(* IEC 61131-3 sources: tianxianzhuantaiPLC/plc/src, 5 files *)

(* ---- Turntable_Constants.st ---- *)
(******************************************************************************
  AutoShop LiteST reference source -- create this as a global constant table.
  Bind only INT wire words to D registers; keep DINT/REAL process values unbound.
******************************************************************************)
VAR_GLOBAL CONSTANT
    (* Modbus wire-register addresses; plc/register-map.md is normative. *)
    D0000_MODE : INT := 0; D0001_DIRECTION : INT := 1;
    D0002_SPEED_INDEX : INT := 2; D0003_START_SEQ : INT := 3;
    D0004_STOP_SEQ : INT := 4; D0005_SET_ZERO_SEQ : INT := 5;
    D0006_RESET_FAULT_SEQ : INT := 6; D0007_POWER_SEQ : INT := 7;
    D0008_HEARTBEAT : INT := 8; D0009_BUFFER_ACK_SEQ : INT := 9;
    D0010_TOTAL_RATIO_HI : INT := 10; D0011_TOTAL_RATIO_LO : INT := 11;
    D0012_ACCEL_HI : INT := 12; D0013_ACCEL_LO : INT := 13;
    D0014_DECEL_HI : INT := 14; D0015_DECEL_LO : INT := 15;
    D0016_STOP_DECEL_HI : INT := 16; D0017_STOP_DECEL_LO : INT := 17;
    D0018_BACKLASH_HI : INT := 18; D0019_BACKLASH_LO : INT := 19;
    D0100_RUN_STATE : INT := 100; D0101_STATUS_FLAGS : INT := 101;
    D0102_FAULT_CODE : INT := 102; D0103_POSITION_HI : INT := 103;
    D0104_POSITION_LO : INT := 104; D0105_TARGET_HI : INT := 105;
    D0106_TARGET_LO : INT := 106; D0107_VELOCITY_HI : INT := 107;
    D0108_VELOCITY_LO : INT := 108; D0109_HEARTBEAT_ECHO : INT := 109;
    D0110_START_ACK_SEQ : INT := 110; D0111_STOP_ACK_SEQ : INT := 111;
    D0112_SET_ZERO_ACK_SEQ : INT := 112; D0113_RESET_FAULT_ACK_SEQ : INT := 113;
    D0114_POWER_ACK_SEQ : INT := 114; D0115_BUFFER_ACKED_SEQ : INT := 115;
    D0116_EVENT_COUNT : INT := 116; D0117_EVENT_GENERATION : INT := 117;
    D0118_RUN_STATUS : INT := 118; D0119_RUN_START_TICK_HI : INT := 119;
    D0120_RUN_START_TICK_LO : INT := 120;
    D0200_PROTOCOL_VERSION : INT := 200; D0201_WORD_ORDER_HI : INT := 201;
    D0202_WORD_ORDER_LO : INT := 202; D0203_TIME_SYNC_REQUEST_SEQ : INT := 203;
    D0204_TICK_HI : INT := 204; D0205_TICK_LO : INT := 205;
    D0206_TIME_SYNC_RESPONSE_SEQ : INT := 206;
    D2000_EVENT_BASE : INT := 2000; D4159_EVENT_END : INT := 4159;

    MODE_MANUAL : INT := 0; MODE_AUTO : INT := 1;
    DIRECTION_CW : INT := 1; DIRECTION_CCW : INT := -1;
    STATE_INITIALIZING : INT := 0; STATE_ZERO_REQUIRED : INT := 1;
    STATE_READY : INT := 2; STATE_MANUAL_RUNNING : INT := 3;
    STATE_AUTO_RUNNING : INT := 4; STATE_STOPPING : INT := 5;
    STATE_AUTO_ABORTED : INT := 6; STATE_FAULT : INT := 7;
    RUN_IDLE : INT := 0; RUN_RUNNING : INT := 1; RUN_COMPLETED : INT := 2;
    RUN_MANUAL_STOPPED : INT := 3; RUN_AUTO_ABORTED : INT := 4;
    RUN_COMMUNICATION_ABORTED : INT := 5; RUN_FAULTED : INT := 6;
    FAULT_NONE : INT := 0; FAULT_INVALID_COMMAND : INT := 1;
    FAULT_ZERO_INTERLOCK : INT := 2; FAULT_AUTO_LIMIT : INT := 3;
    FAULT_MOTION : INT := 4; FAULT_POSITION_READ : INT := 5;
    FAULT_VELOCITY_READ : INT := 6; FAULT_HEARTBEAT : INT := 7;
    FAULT_STOP_UNSAFE : INT := 8; FAULT_AXIS_CONFIG : INT := 9;
    FAULT_START_REJECTED : INT := 10; FAULT_RESET : INT := 11;

    STATUS_ZERO_VALID : INT := 1; STATUS_POWERED : INT := 2;
    STATUS_SOFT_LIMIT : INT := 4; STATUS_BUFFER_READY : INT := 8;
    STATUS_HEARTBEAT_OK : INT := 16;
    PROTOCOL_VERSION : INT := 2;
    WORD_ORDER_PROBE_HIGH : INT := 4660; WORD_ORDER_PROBE_LOW : INT := 22136;
    TOTAL_RATIO_MILLI : DINT := 50000; (* 50.000:1 *)
    SPEED_1_DEG_S : REAL := 1.0; SPEED_2_DEG_S : REAL := 2.0;
    SPEED_3_DEG_S : REAL := 4.0; SPEED_4_DEG_S : REAL := 5.0;
    SPEED_5_DEG_S : REAL := 10.0;
    ACCELERATION_DEG_S2 : REAL := 5.0; DECELERATION_DEG_S2 : REAL := 5.0;
    SOFTWARE_STOP_DECEL_DEG_S2 : REAL := 10.0;
    ACCELERATION_MILLI_DEG_S2 : DINT := 5000;
    DECELERATION_MILLI_DEG_S2 : DINT := 5000;
    SOFTWARE_STOP_DECEL_MILLI_DEG_S2 : DINT := 10000;
    SOFT_LIMIT_MIN_DEG : REAL := -360.0; SOFT_LIMIT_MAX_DEG : REAL := 360.0;
    AUTO_DISTANCE_DEG : REAL := 360.0;
    HEARTBEAT_TIMEOUT_SCANS : INT := 1000;
    EVENT_CAPACITY : INT := 360; EVENT_RECORD_WORDS : INT := 6;
    EVENT_WORD_COUNT : INT := 2160; EVENT_MAX_CROSSINGS_PER_SCAN : INT := 360;
END_VAR

(* Create this as the sole global MODBUS_D variable table and bind addresses
   here. PRG_MAIN consumes these globals; do not redeclare them locally. *)
VAR_GLOBAL
    iD0000Mode, iD0001Direction, iD0002SpeedIndex : INT;
    iD0003StartSeq, iD0004StopSeq, iD0005SetZeroSeq, iD0006ResetFaultSeq : INT;
    iD0007PowerSeq, iD0008Heartbeat, iD0009BufferAckSeq : INT;
    iD0010RatioHi, iD0011RatioLo, iD0012AccelHi, iD0013AccelLo : INT;
    iD0014DecelHi, iD0015DecelLo, iD0016StopDecelHi, iD0017StopDecelLo : INT;
    iD0018BacklashHi, iD0019BacklashLo : INT;
    iD0100RunState, iD0101StatusFlags, iD0102FaultCode : INT;
    iD0103PositionHi, iD0104PositionLo, iD0105TargetHi, iD0106TargetLo : INT;
    iD0107VelocityHi, iD0108VelocityLo, iD0109HeartbeatEcho : INT;
    iD0110StartAck, iD0111StopAck, iD0112SetZeroAck, iD0113ResetFaultAck : INT;
    iD0114PowerAck, iD0115BufferAcked, iD0116EventCount, iD0117Generation : INT;
    iD0118RunStatus, iD0119RunStartTickHi, iD0120RunStartTickLo : INT;
    iD0200ProtocolVersion, iD0201WordOrderHi, iD0202WordOrderLo : INT;
    iD0203TimeSyncRequest, iD0204TickHi, iD0205TickLo, iD0206TimeSyncResponse : INT;
    aD2000Events : ARRAY[0..2159] OF INT;
END_VAR

(* ---- Turntable_RegisterCodec.st ---- *)
(******************************************************************************
  AutoShop LiteST reference source -- create these two FCs before the FBs.
  DINT values are always explicitly represented as high-word then low-word INTs.
  Read and verify D0201:D0202 (0x1234/0x5678) on the actual PLC before any
  hardware write.  Do not rely on a native DINT variable-table binding order.
******************************************************************************)
FUNCTION FC_DecodeI32 : DINT
VAR_INPUT
    iHighWord : INT;
    iLowWord : INT;
END_VAR
VAR
    diLowWord : DINT;
END_VAR
diLowWord := INT_TO_DINT(iLowWord);
IF diLowWord < 0 THEN diLowWord := diLowWord + 65536; END_IF;
FC_DecodeI32 := INT_TO_DINT(iHighWord) * 65536 + diLowWord;
END_FUNCTION

FUNCTION FC_SplitI32 : BOOL
VAR_INPUT
    diValue : DINT;
END_VAR
VAR_OUTPUT
    iHighWord : INT;
    iLowWord : INT;
END_VAR
VAR
    diHighWord : DINT;
    diLowWord : DINT;
END_VAR
diHighWord := diValue / 65536;
diLowWord := diValue MOD 65536;
IF diLowWord < 0 THEN
    diLowWord := diLowWord + 65536;
    diHighWord := diHighWord - 1;
END_IF;
IF diHighWord >= 32768 THEN diHighWord := diHighWord - 65536; END_IF;
IF diLowWord >= 32768 THEN diLowWord := diLowWord - 65536; END_IF;
iHighWord := DINT_TO_INT(diHighWord);
iLowWord := DINT_TO_INT(diLowWord);
FC_SplitI32 := TRUE;
END_FUNCTION

FUNCTION FC_SplitU32 : BOOL
VAR_INPUT
    diValue : DINT;
END_VAR
VAR_OUTPUT
    iHighWord : INT;
    iLowWord : INT;
END_VAR
VAR
    diHighWord : DINT;
    diLowWord : DINT;
END_VAR
diHighWord := diValue / 65536;
diLowWord := diValue MOD 65536;
IF diLowWord < 0 THEN
    diLowWord := diLowWord + 65536;
    diHighWord := diHighWord - 1;
END_IF;
IF diHighWord >= 32768 THEN diHighWord := diHighWord - 65536; END_IF;
IF diLowWord >= 32768 THEN diLowWord := diLowWord - 65536; END_IF;
iHighWord := DINT_TO_INT(diHighWord);
iLowWord := DINT_TO_INT(diLowWord);
FC_SplitU32 := TRUE;
END_FUNCTION

(* ---- FB_DegreeLogger.st ---- *)
(******************************************************************************
  AutoShop LiteST reference source -- create FB_DegreeLogger, paste declaration
  and body.  aEventWords is the INT[2160] variable-table array bound at D2000.
******************************************************************************)
FUNCTION_BLOCK FB_DegreeLogger
VAR_INPUT
    rPreviousPositionDeg : REAL;
    rCurrentPositionDeg : REAL;
    rRunOriginDeg : REAL;
    iDirection : INT;
    udiRunStartTickMs : UDINT;
    udiNowTickMs : UDINT;
    bRunStarted : BOOL;
    bRunFinished : BOOL;
    bBufferAckEdge : BOOL;
END_VAR
VAR_IN_OUT
    aEventWords : ARRAY[0..2159] OF INT;
END_VAR
VAR_OUTPUT
    bBufferReady : BOOL;
    uiEventCount : UINT;
    uiGeneration : UINT;
END_VAR
VAR
    rPreviousTravel : REAL;
    rCurrentTravel : REAL;
    rCrossingPosition : REAL;
    iFirstAngle : INT;
    iLastAngle : INT;
    iCrossing : INT;
    iTravelAngle : INT;
    iBase : INT;
    diPositionMdeg : DINT;
    udiElapsedMs : UDINT;
    iPositionHigh : INT;
    iPositionLow : INT;
    iElapsedHigh : INT;
    iElapsedLow : INT;
END_VAR

(* An acknowledged completed buffer is released before a possible run start. *)
IF bBufferAckEdge AND bBufferReady THEN
    bBufferReady := FALSE;
    uiEventCount := 0;
END_IF;

IF bRunStarted AND NOT bBufferReady THEN
    uiEventCount := 0;
    uiGeneration := uiGeneration + 1;
END_IF;

(* A sealed buffer is immutable. A controller prevents another run until ACK. *)
IF NOT bBufferReady AND NOT bRunStarted THEN
    rPreviousTravel := (rPreviousPositionDeg - rRunOriginDeg) * REAL(iDirection);
    rCurrentTravel := (rCurrentPositionDeg - rRunOriginDeg) * REAL(iDirection);
    iFirstAngle := MAX(1, REAL_TO_INT(FLOOR(rPreviousTravel)) + 1);
    iLastAngle := MIN(360, REAL_TO_INT(FLOOR(rCurrentTravel)));

    (* Fixed guard: at most 360 legal travel-angle writes per scan. *)
    FOR iCrossing := 1 TO 360 DO
        iTravelAngle := iFirstAngle + iCrossing - 1;
        IF iTravelAngle > iLastAngle THEN
            EXIT;
        END_IF;
        IF uiEventCount < 360 THEN
            iBase := 6 * uiEventCount;
            rCrossingPosition := rRunOriginDeg + REAL(iDirection) * REAL(iTravelAngle);
            diPositionMdeg := REAL_TO_DINT(rCrossingPosition * 1000.0);
            (* UDINT subtraction intentionally handles the 49.7-day tick wrap. *)
            udiElapsedMs := udiNowTickMs - udiRunStartTickMs;
            FC_SplitI32(diValue := diPositionMdeg, iHighWord => iPositionHigh, iLowWord => iPositionLow);
            FC_SplitU32(udiValue := udiElapsedMs, iHighWord => iElapsedHigh, iLowWord => iElapsedLow);
            aEventWords[iBase + 0] := INT(uiEventCount + 1);
            aEventWords[iBase + 1] := iTravelAngle;
            aEventWords[iBase + 2] := iPositionHigh;
            aEventWords[iBase + 3] := iPositionLow;
            aEventWords[iBase + 4] := iElapsedHigh;
            aEventWords[iBase + 5] := iElapsedLow;
            uiEventCount := uiEventCount + 1;
        ELSE
            EXIT;
        END_IF;
    END_FOR;
END_IF;

IF bRunFinished THEN
    bBufferReady := TRUE;
END_IF;
END_FUNCTION_BLOCK

(* ---- FB_TurntableControl.st ---- *)
(******************************************************************************
  AutoShop LiteST reference -- create FB_TurntableControl then paste it.
  It is deterministic: a commanded move remains active until MC_Stop confirms
  standstill. The heartbeat is a communication watchdog, not safety-rated.
******************************************************************************)
FUNCTION_BLOCK FB_TurntableControl
VAR_INPUT
    uiMode : UINT; iDirection : INT; uiSpeedIndex : UINT;
    uiStartSeq : UINT; uiStopSeq : UINT; uiSetZeroSeq : UINT;
    uiResetFaultSeq : UINT; uiPowerSeq : UINT; uiHeartbeat : UINT;
    uiBufferAckSeq : UINT; udiNowTickMs : UDINT;
    diTotalRatioMilli : DINT; diRequestedAccelMilli : DINT;
    diRequestedDecelMilli : DINT; diRequestedStopDecelMilli : DINT;
    diBacklashMilli : DINT;
    rActualPositionDeg : REAL; rActualVelocityDegS : REAL;
    bPositionValid : BOOL; bVelocityValid : BOOL;
    bPositionReadError : BOOL; bVelocityReadError : BOOL;
    bPowerStatus : BOOL; bPowerError : BOOL; bMoveDone : BOOL;
    bMoveBusy : BOOL; bMoveAborted : BOOL; bMoveError : BOOL;
    bStopDone : BOOL; bStopBusy : BOOL; bStopError : BOOL;
    bSetPositionDone : BOOL; bSetPositionError : BOOL;
    bResetDone : BOOL; bResetBusy : BOOL; bResetError : BOOL;
    bLoggerBufferReady : BOOL; uiLoggerEventCount : UINT;
END_VAR
VAR_OUTPUT
    bPowerEnable : BOOL; bMoveRequest : BOOL; bStopRequest : BOOL;
    bSetZeroRequest : BOOL; bResetRequest : BOOL;
    bRunStarted : BOOL; bRunFinished : BOOL; bBufferAckEdge : BOOL;
    rMoveDistance : REAL; rSelectedVelocity : REAL;
    rAcceleration : REAL; rDeceleration : REAL; rStopDeceleration : REAL;
    rRunOriginDeg : REAL; iRunDirection : INT; udiRunStartTickMs : UDINT;
    rAcceptedTargetDeg : REAL;
    uiRunState : UINT; uiRunStatus : UINT; uiFaultCode : UINT;
    uiStatusFlags : UINT; uiHeartbeatEcho : UINT;
    uiStartAckSeq : UINT; uiStopAckSeq : UINT; uiSetZeroAckSeq : UINT;
    uiResetFaultAckSeq : UINT; uiPowerAckSeq : UINT; uiBufferAckedSeq : UINT;
    uiRetainedStopReason : UINT; bUnsafeStopFailure : BOOL;
END_VAR
VAR RETAIN
    bZeroValid : BOOL;
    uiRetainedStopReasonNv : UINT;
END_VAR
VAR
    uiLastHeartbeat : UINT; uiHeartbeatAgeScans : UINT;
    bActiveRun : BOOL; bStopLatched : BOOL; bFaultStopPending : BOOL;
    uiPendingFaultCode : UINT; bPowerCommandValue : BOOL;
    bResetPending : BOOL; uiResetPendingSeq : UINT;
    bStartAccepted : BOOL;
    rCandidateTargetDeg : REAL;
END_VAR

(* Defaults are one-scan rising-edge request pulses. *)
bMoveRequest := FALSE; bStopRequest := FALSE; bSetZeroRequest := FALSE;
bResetRequest := FALSE; bRunStarted := FALSE; bRunFinished := FALSE;
bBufferAckEdge := FALSE;

IF uiRunState = STATE_INITIALIZING THEN
    IF bZeroValid THEN uiRunState := STATE_READY; ELSE uiRunState := STATE_ZERO_REQUIRED; END_IF;
END_IF;

IF uiHeartbeat <> uiLastHeartbeat THEN
    uiLastHeartbeat := uiHeartbeat; uiHeartbeatAgeScans := 0; uiHeartbeatEcho := uiHeartbeat;
ELSIF uiHeartbeatAgeScans < 65535 THEN
    uiHeartbeatAgeScans := uiHeartbeatAgeScans + 1;
END_IF;

(* Terminal Stop response is handled before accepting another command. *)
IF bStopError AND bStopLatched THEN
    (* Unsafe terminal path: motion stop was not confirmed. Inhibit power and
       keep the event buffer unsealed for on-site assessment; do not auto-retry. *)
    bActiveRun := FALSE; bStopLatched := FALSE; bUnsafeStopFailure := TRUE;
    uiRunState := STATE_FAULT; uiRunStatus := RUN_FAULTED; uiFaultCode := FAULT_STOP_UNSAFE;
    uiRetainedStopReason := RUN_FAULTED; uiRetainedStopReasonNv := RUN_FAULTED;
ELSIF bStopDone AND bActiveRun THEN
    bActiveRun := FALSE; bStopLatched := FALSE; bRunFinished := TRUE;
    IF bFaultStopPending THEN
        bFaultStopPending := FALSE; uiRunState := STATE_FAULT; uiRunStatus := RUN_FAULTED;
        uiFaultCode := uiPendingFaultCode; rAcceptedTargetDeg := rActualPositionDeg;
    ELSE
        uiRunState := STATE_READY; uiRunStatus := uiRetainedStopReason;
        rAcceptedTargetDeg := rActualPositionDeg;
    END_IF;
END_IF;

(* RESET is an axis instruction result, not a display-only flag clear. *)
IF bResetPending AND (bResetDone OR bResetError) THEN
    uiResetFaultAckSeq := uiResetPendingSeq; bResetPending := FALSE;
    IF bResetDone THEN
        uiFaultCode := FAULT_NONE; uiRunStatus := RUN_IDLE;
        bFaultStopPending := FALSE; uiPendingFaultCode := FAULT_NONE;
        bStopLatched := FALSE; bUnsafeStopFailure := FALSE;
        uiRetainedStopReason := RUN_IDLE; uiRetainedStopReasonNv := RUN_IDLE;
        IF bZeroValid THEN uiRunState := STATE_READY; ELSE uiRunState := STATE_ZERO_REQUIRED; END_IF;
    ELSE
        uiRunState := STATE_FAULT; uiRunStatus := RUN_FAULTED; uiFaultCode := FAULT_RESET;
    END_IF;
END_IF;

(* STOP_SEQ is first and also consumes a same/earlier START_SEQ. *)
IF uiStopSeq <> uiStopAckSeq THEN
    uiStopAckSeq := uiStopSeq;
    uiStartAckSeq := uiStartSeq; (* discard pending start; stop has priority *)
    IF bActiveRun AND NOT bStopLatched THEN
        bStopLatched := TRUE; bStopRequest := TRUE; uiRunState := STATE_STOPPING;
        IF uiMode = MODE_AUTO THEN uiRetainedStopReason := RUN_AUTO_ABORTED;
        ELSE uiRetainedStopReason := RUN_MANUAL_STOPPED; END_IF;
        uiRetainedStopReasonNv := uiRetainedStopReason; uiRunStatus := uiRetainedStopReason;
    END_IF;
ELSIF bActiveRun AND NOT bStopLatched AND
      (bPositionReadError OR bVelocityReadError OR NOT bPositionValid OR NOT bVelocityValid
       OR bPowerError OR bMoveError OR bMoveAborted) THEN
    (* Preserve active motion and command MC_Stop in this scan; only Done seals it. *)
    bStopLatched := TRUE; bFaultStopPending := TRUE; bStopRequest := TRUE;
    uiRunState := STATE_STOPPING; uiRunStatus := RUN_FAULTED;
    uiRetainedStopReason := RUN_FAULTED; uiRetainedStopReasonNv := RUN_FAULTED;
    IF bPositionReadError OR NOT bPositionValid THEN uiPendingFaultCode := FAULT_POSITION_READ;
    ELSIF bVelocityReadError OR NOT bVelocityValid THEN uiPendingFaultCode := FAULT_VELOCITY_READ;
    ELSE uiPendingFaultCode := FAULT_MOTION; END_IF;
ELSIF bActiveRun AND NOT bStopLatched AND (uiHeartbeatAgeScans > 1000) THEN
    bStopLatched := TRUE; bStopRequest := TRUE; uiRunState := STATE_STOPPING;
    uiRetainedStopReason := RUN_COMMUNICATION_ABORTED;
    uiRetainedStopReasonNv := uiRetainedStopReason; uiRunStatus := RUN_COMMUNICATION_ABORTED;
    uiFaultCode := FAULT_HEARTBEAT;
ELSIF uiResetFaultSeq <> uiResetFaultAckSeq AND NOT bResetPending THEN
    IF bActiveRun THEN
        uiResetFaultAckSeq := uiResetFaultSeq; uiFaultCode := FAULT_INVALID_COMMAND;
    ELSE
        bResetPending := TRUE; uiResetPendingSeq := uiResetFaultSeq; bResetRequest := TRUE;
    END_IF;
ELSIF uiBufferAckSeq <> uiBufferAckedSeq THEN
    IF NOT bActiveRun THEN uiBufferAckedSeq := uiBufferAckSeq; bBufferAckEdge := TRUE; END_IF;
ELSIF uiPowerSeq <> uiPowerAckSeq THEN
    uiPowerAckSeq := uiPowerSeq;
    IF NOT bActiveRun THEN bPowerCommandValue := NOT bPowerCommandValue; END_IF;
ELSIF uiSetZeroSeq <> uiSetZeroAckSeq THEN
    IF NOT bActiveRun AND NOT bMoveBusy AND NOT bStopBusy AND NOT bPowerError
       AND bPositionValid AND ABS(rActualVelocityDegS) < 0.001 THEN
        uiSetZeroAckSeq := uiSetZeroSeq; bSetZeroRequest := TRUE;
    ELSE
        uiSetZeroAckSeq := uiSetZeroSeq; uiFaultCode := FAULT_INVALID_COMMAND;
    END_IF;
ELSIF uiStartSeq <> uiStartAckSeq THEN
    (* Every START_SEQ receives a final accept or reject acknowledgement. *)
    uiStartAckSeq := uiStartSeq; bStartAccepted := TRUE;
    IF bActiveRun OR bLoggerBufferReady OR NOT bZeroValid OR NOT bPowerStatus
       OR NOT bPositionValid OR NOT bVelocityValid OR bPowerError OR bMoveError
       OR bUnsafeStopFailure OR (uiHeartbeatAgeScans > 1000) THEN bStartAccepted := FALSE; END_IF;
    IF (diRequestedAccelMilli <= 0) OR (diRequestedDecelMilli <= 0)
       OR (diRequestedStopDecelMilli <= 0) OR (diBacklashMilli <> 0)
       OR (diTotalRatioMilli <> TOTAL_RATIO_MILLI) THEN bStartAccepted := FALSE; END_IF;
    CASE uiSpeedIndex OF
        1: rSelectedVelocity := 1.0; 2: rSelectedVelocity := 2.0;
        3: rSelectedVelocity := 4.0; 4: rSelectedVelocity := 5.0;
        5: rSelectedVelocity := 10.0;
    ELSE bStartAccepted := FALSE; rSelectedVelocity := 0.0;
    END_CASE;
    IF (iDirection <> DIRECTION_CW) AND (iDirection <> DIRECTION_CCW) THEN bStartAccepted := FALSE; END_IF;
    IF uiMode = MODE_AUTO THEN
        rCandidateTargetDeg := rActualPositionDeg + 360.0 * REAL(iDirection);
        IF (rCandidateTargetDeg < -360.0) OR (rCandidateTargetDeg > 360.0) THEN bStartAccepted := FALSE; END_IF;
    ELSIF uiMode = MODE_MANUAL THEN
        rCandidateTargetDeg := rActualPositionDeg + 360.0 * REAL(iDirection);
        IF rCandidateTargetDeg > 360.0 THEN rCandidateTargetDeg := 360.0; END_IF;
        IF rCandidateTargetDeg < -360.0 THEN rCandidateTargetDeg := -360.0; END_IF;
    ELSE bStartAccepted := FALSE;
    END_IF;
    rMoveDistance := rCandidateTargetDeg - rActualPositionDeg;
    IF ABS(rMoveDistance) < 0.001 THEN bStartAccepted := FALSE; END_IF;
    IF bStartAccepted THEN
        (* Parameters are validated and latched only at accepted-run boundary. *)
        uiFaultCode := FAULT_NONE; bFaultStopPending := FALSE;
        uiPendingFaultCode := FAULT_NONE; bStopLatched := FALSE;
        uiRetainedStopReason := RUN_IDLE; uiRetainedStopReasonNv := RUN_IDLE;
        rAcceleration := DINT_TO_REAL(diRequestedAccelMilli) / 1000.0;
        rDeceleration := DINT_TO_REAL(diRequestedDecelMilli) / 1000.0;
        rStopDeceleration := DINT_TO_REAL(diRequestedStopDecelMilli) / 1000.0;
        rAcceptedTargetDeg := rCandidateTargetDeg;
        bMoveRequest := TRUE; bRunStarted := TRUE; bActiveRun := TRUE; bStopLatched := FALSE;
        rRunOriginDeg := rActualPositionDeg; iRunDirection := iDirection; udiRunStartTickMs := udiNowTickMs;
        uiRunStatus := RUN_RUNNING;
        IF uiMode = MODE_AUTO THEN uiRunState := STATE_AUTO_RUNNING; ELSE uiRunState := STATE_MANUAL_RUNNING; END_IF;
    ELSE
        uiFaultCode := FAULT_START_REJECTED; uiRunStatus := RUN_FAULTED;
        IF NOT bZeroValid THEN uiRunState := STATE_ZERO_REQUIRED; ELSE uiRunState := STATE_FAULT; END_IF;
    END_IF;
END_IF;

IF bSetPositionDone THEN bZeroValid := TRUE; IF NOT bActiveRun THEN uiRunState := STATE_READY; END_IF; END_IF;
IF bSetPositionError THEN uiRunState := STATE_FAULT; uiRunStatus := RUN_FAULTED; uiFaultCode := FAULT_MOTION; END_IF;
IF bMoveDone AND bActiveRun AND NOT bStopLatched THEN
    bActiveRun := FALSE; bRunFinished := TRUE; uiRunState := STATE_READY; uiRunStatus := RUN_COMPLETED;
END_IF;

bPowerEnable := bPowerCommandValue AND NOT bUnsafeStopFailure;
uiStatusFlags := 0;
IF bZeroValid THEN uiStatusFlags := uiStatusFlags OR STATUS_ZERO_VALID; END_IF;
IF bPowerStatus THEN uiStatusFlags := uiStatusFlags OR STATUS_POWERED; END_IF;
IF bLoggerBufferReady THEN uiStatusFlags := uiStatusFlags OR STATUS_BUFFER_READY; END_IF;
IF uiHeartbeatAgeScans <= 1000 THEN uiStatusFlags := uiStatusFlags OR STATUS_HEARTBEAT_OK; END_IF;
IF (rActualPositionDeg <= -360.0) OR (rActualPositionDeg >= 360.0) THEN uiStatusFlags := uiStatusFlags OR STATUS_SOFT_LIMIT; END_IF;
END_FUNCTION_BLOCK

(* ---- PRG_MAIN.st ---- *)
(******************************************************************************
  AutoShop LiteST reference source -- create program POU PRG_MAIN and paste the
  declaration/body. Create Axis_0 in AutoShop's axis configuration, not here.
  Create the MODBUS_D variable table described in plc/README.md before binding.
******************************************************************************)
PROGRAM PRG_MAIN
VAR
    udiPlcTickMs : UDINT;
    rActualPosition, rActualVelocity : REAL;
    rMoveDistance, rSelectedVelocity, rAcceleration, rDeceleration, rStopDeceleration : REAL;
    bPowerEnable, bPowerStatus, bPowerBusy, bPowerError : BOOL;
    iPowerErrorID : INT;
    bSetPositionExecute, bSetPositionDone, bSetPositionBusy, bSetPositionError : BOOL;
    iSetPositionErrorID : INT;
    bMoveExecute, bMoveDone, bMoveBusy, bMoveAborted, bMoveError : BOOL;
    iMoveErrorID : INT;
    bStopExecute, bStopDone, bStopBusy, bStopError : BOOL;
    iStopErrorID : INT;
    bResetExecute, bResetDone, bResetBusy, bResetError : BOOL;
    iResetErrorID : INT;
    bPositionValid, bPositionBusy, bPositionError : BOOL;
    iPositionErrorID : INT;
    bVelocityValid, bVelocityBusy, bVelocityError : BOOL;
    iVelocityErrorID : INT;
    rPreviousPosition : REAL;
    rLoggerPosition : REAL;
    bLoggerStarted, bLoggerFinished, bLoggerAck : BOOL;
    bLoggerBufferReady : BOOL;
    uiLoggerEventCount, uiLoggerGeneration : UINT;
    diPositionMdeg, diTargetMdeg, diVelocityMdegS : DINT;
    diTotalRatioMilli, diRequestedAccelMilli, diRequestedDecelMilli : DINT;
    diRequestedStopDecelMilli, diBacklashMilli : DINT;
    fbControl : FB_TurntableControl;
    fbLogger : FB_DegreeLogger;
END_VAR

(* PRG_MAIN must be scheduled as a constant 1 ms task; tick is not retained. *)
udiPlcTickMs := udiPlcTickMs + 1;

(* Decode all runtime parameters explicitly. D1010 ratio must match the
   offline Axis_0 scaling; phase 1 does not perform backlash compensation. *)
diTotalRatioMilli := FC_DecodeI32(iHighWord := iD1010RatioHi, iLowWord := iD1011RatioLo);
diRequestedAccelMilli := FC_DecodeI32(iHighWord := iD1012AccelHi, iLowWord := iD1013AccelLo);
diRequestedDecelMilli := FC_DecodeI32(iHighWord := iD1014DecelHi, iLowWord := iD1015DecelLo);
diRequestedStopDecelMilli := FC_DecodeI32(iHighWord := iD1016StopDecelHi, iLowWord := iD1017StopDecelLo);
diBacklashMilli := FC_DecodeI32(iHighWord := iD1018BacklashHi, iLowWord := iD1019BacklashLo);

(* 1. Refresh feedback first. These enables remain TRUE for continuously valid reads. *)
MC_ReadActualPosition(Enable := TRUE, Axis := Axis_0,
    Valid => bPositionValid, Busy => bPositionBusy,
    Position => rActualPosition,
    Error => bPositionError, ErrorID => iPositionErrorID);

MC_ReadActualVelocity(Enable := TRUE, Axis := Axis_0,
    Valid => bVelocityValid, Busy => bVelocityBusy,
    Velocity => rActualVelocity,
    Error => bVelocityError, ErrorID => iVelocityErrorID);

(* Invalid position feedback must not create synthetic degree crossings. *)
IF bPositionValid AND NOT bPositionError THEN
    rLoggerPosition := rActualPosition;
END_IF;

(* 2. Deterministic command/state decision uses current feedback and raw INT wire words. *)
fbControl(
    uiMode := UINT(iD1000Mode), iDirection := iD1001Direction,
    uiSpeedIndex := UINT(iD1002SpeedIndex), uiStartSeq := UINT(iD1003StartSeq),
    uiStopSeq := UINT(iD1004StopSeq), uiSetZeroSeq := UINT(iD1005SetZeroSeq),
    uiResetFaultSeq := UINT(iD1006ResetFaultSeq), uiPowerSeq := UINT(iD1007PowerSeq),
    uiHeartbeat := UINT(iD1008Heartbeat), uiBufferAckSeq := UINT(iD1009BufferAckSeq),
    udiNowTickMs := udiPlcTickMs,
    diTotalRatioMilli := diTotalRatioMilli, diRequestedAccelMilli := diRequestedAccelMilli,
    diRequestedDecelMilli := diRequestedDecelMilli, diRequestedStopDecelMilli := diRequestedStopDecelMilli,
    diBacklashMilli := diBacklashMilli,
    rActualPositionDeg := rActualPosition, rActualVelocityDegS := rActualVelocity,
    bPositionValid := bPositionValid, bVelocityValid := bVelocityValid,
    bPositionReadError := bPositionError, bVelocityReadError := bVelocityError,
    bPowerStatus := bPowerStatus, bPowerError := bPowerError, bMoveDone := bMoveDone,
    bMoveBusy := bMoveBusy, bMoveAborted := bMoveAborted, bMoveError := bMoveError,
    bStopDone := bStopDone, bStopBusy := bStopBusy, bStopError := bStopError,
    bSetPositionDone := bSetPositionDone, bSetPositionError := bSetPositionError,
    bResetDone := bResetDone, bResetBusy := bResetBusy, bResetError := bResetError,
    bLoggerBufferReady := bLoggerBufferReady, uiLoggerEventCount := uiLoggerEventCount);

bPowerEnable := fbControl.bPowerEnable;
rMoveDistance := fbControl.rMoveDistance; rSelectedVelocity := fbControl.rSelectedVelocity;
rAcceleration := fbControl.rAcceleration; rDeceleration := fbControl.rDeceleration;
rStopDeceleration := fbControl.rStopDeceleration;

(* 3. Rising-edge commands. Motion parameters latch on Execute's rising edge. *)
bSetPositionExecute := fbControl.bSetZeroRequest;
MC_SetPosition(Execute := bSetPositionExecute, Axis := Axis_0,
    Position := 0.0, Mode := 0,
    Done => bSetPositionDone, Busy => bSetPositionBusy,
    Error => bSetPositionError, ErrorID => iSetPositionErrorID);
bSetPositionExecute := FALSE;

bResetExecute := fbControl.bResetRequest;
MC_Reset(Execute := bResetExecute, Axis := Axis_0,
    Done => bResetDone, Busy => bResetBusy,
    Error => bResetError, ErrorID => iResetErrorID);
bResetExecute := FALSE;

bMoveExecute := fbControl.bMoveRequest;
MC_MoveRelative(Execute := bMoveExecute, Axis := Axis_0,
    Distance := rMoveDistance, Velocity := rSelectedVelocity,
    Acceleration := rAcceleration, Deceleration := rDeceleration,
    CurveType := 0, Done => bMoveDone, Busy => bMoveBusy,
    CommandAborted => bMoveAborted,
    Error => bMoveError, ErrorID => iMoveErrorID);
bMoveExecute := FALSE;

IF fbControl.bStopRequest THEN
    bStopExecute := TRUE;
END_IF;
(* MC_ImmediateStop is not used: this is a controlled software deceleration. *)
MC_Stop(Execute := bStopExecute, Axis := Axis_0,
    Deceleration := rStopDeceleration, CurveType := 0,
    Done => bStopDone, Busy => bStopBusy,
    Error => bStopError, ErrorID => iStopErrorID);
(* Done with Execute TRUE holds Stopping; reset only after Done permits Standstill. *)
IF bStopDone OR bStopError THEN
    bStopExecute := FALSE;
END_IF;

MC_Power(Enable := bPowerEnable, Axis := Axis_0,
    Status => bPowerStatus, Busy => bPowerBusy,
    Error => bPowerError, ErrorID => iPowerErrorID);

(* 4. Capture all crossed travel integers, then publish a stable register snapshot. *)
bLoggerStarted := fbControl.bRunStarted; bLoggerFinished := fbControl.bRunFinished;
bLoggerAck := fbControl.bBufferAckEdge;
fbLogger(rPreviousPositionDeg := rPreviousPosition, rCurrentPositionDeg := rLoggerPosition,
    rRunOriginDeg := fbControl.rRunOriginDeg, iDirection := fbControl.iRunDirection,
    udiRunStartTickMs := fbControl.udiRunStartTickMs, udiNowTickMs := udiPlcTickMs,
    bRunStarted := bLoggerStarted, bRunFinished := bLoggerFinished, bBufferAckEdge := bLoggerAck,
    aEventWords := aD2000Events, bBufferReady => bLoggerBufferReady,
    uiEventCount => uiLoggerEventCount, uiGeneration => uiLoggerGeneration);
IF bPositionValid AND NOT bPositionError THEN
    rPreviousPosition := rLoggerPosition;
END_IF;

iD1100RunState := INT(fbControl.uiRunState); iD1101StatusFlags := INT(fbControl.uiStatusFlags);
iD1102FaultCode := INT(fbControl.uiFaultCode); iD1109HeartbeatEcho := INT(fbControl.uiHeartbeatEcho);
iD1110StartAck := INT(fbControl.uiStartAckSeq); iD1111StopAck := INT(fbControl.uiStopAckSeq);
iD1112SetZeroAck := INT(fbControl.uiSetZeroAckSeq); iD1113ResetFaultAck := INT(fbControl.uiResetFaultAckSeq);
iD1114PowerAck := INT(fbControl.uiPowerAckSeq); iD1115BufferAcked := INT(fbControl.uiBufferAckedSeq);
iD1116EventCount := INT(uiLoggerEventCount); iD1117Generation := INT(uiLoggerGeneration);
iD1118RunStatus := INT(fbControl.uiRunStatus); iD1200ProtocolVersion := INT(PROTOCOL_VERSION);
iD1201WordOrderHi := WORD_ORDER_PROBE_HIGH; iD1202WordOrderLo := WORD_ORDER_PROBE_LOW;
iD1206TimeSyncResponse := iD1203TimeSyncRequest;

diPositionMdeg := REAL_TO_DINT(rActualPosition * 1000.0);
diTargetMdeg := REAL_TO_DINT(fbControl.rAcceptedTargetDeg * 1000.0);
diVelocityMdegS := REAL_TO_DINT(rActualVelocity * 1000.0);
FC_SplitI32(diValue := diPositionMdeg, iHighWord => iD1103PositionHi, iLowWord => iD1104PositionLo);
FC_SplitI32(diValue := diTargetMdeg, iHighWord => iD1105TargetHi, iLowWord => iD1106TargetLo);
FC_SplitI32(diValue := diVelocityMdegS, iHighWord => iD1107VelocityHi, iLowWord => iD1108VelocityLo);
FC_SplitU32(udiValue := udiPlcTickMs, iHighWord => iD1204TickHi, iLowWord => iD1205TickLo);
END_PROGRAM
